//==================================================================================================
//								RJM Maszyny sp. z o.o.
//									04.02.2022
//	Obsługa elektrozaworu 5/3 odpowietrzony w pozycji środkowej
// 	v1.0	|| TC v 3.1.4024.22		|| - pierwsza wersja
//==================================================================================================
FUNCTION_BLOCK FB_Elektrozawor_5na3_Odpowietrzony IMPLEMENTS I_Elektrozawor_5na
VAR
	fbCewkaA								: FB_ElektrozaworCewka;
	fbCewkaB								: FB_ElektrozaworCewka;
END_VAR

//==================================================================================================
//								RJM Maszyny sp. z o.o.
//									04.02.2022
//	Włączenie cewki - wyjscie 2
// 	v1.0	|| TC v 3.1.4024.22		|| - pierwsza wersja
//==================================================================================================METHOD WlaczWyjscie2 : BOOL
VAR_INPUT
END_VAR
fbCewkaA.Wlacz ();
END_METHOD

//==================================================================================================
//								RJM Maszyny sp. z o.o.
//									04.02.2022
//	Włączenie cewki - wyjscie 4
// 	v1.0	|| TC v 3.1.4024.22		|| - pierwsza wersja
//==================================================================================================
METHOD WlaczWyjscie4 : BOOL
VAR_INPUT
END_VAR
fbCewkaB.Wlacz ();
END_METHOD

//==================================================================================================
//								RJM Maszyny sp. z o.o.
//									04.02.2022
//	Wyłączenie cewki - wyjscie 2
// 	v1.0	|| TC v 3.1.4024.22		|| - pierwsza wersja
//==================================================================================================METHOD WylaczWyjscie2 : BOOL
VAR_INPUT
END_VAR
fbCewkaA.Wylacz ();
END_METHOD

//==================================================================================================
//								RJM Maszyny sp. z o.o.
//									04.02.2022
//	Wyłączenie cewki - wyjscie 4
// 	v1.0	|| TC v 3.1.4024.22		|| - pierwsza wersja
//==================================================================================================
METHOD WylaczWyjscie4 : BOOL
VAR_INPUT
END_VAR
fbCewkaB.Wylacz ();
END_METHOD

END_FUNCTION_BLOCK

(* stored: Version 1.1.0.1, ProductVersion 3.1.4024.11
   POU FB_Elektrozawor_5na3_Odpowietrzony: Id {f17b99e1-6967-4370-8cd2-c2384288e58c}, SpecialFunc None
   Method WlaczWyjscie2: Id {05977016-e664-463d-87c0-181849a20e65}
   Method WlaczWyjscie4: Id {cc4e5290-0150-4cef-b5cd-45f8eb479fdd}
   Method WylaczWyjscie2: Id {6db52a01-b744-4f16-808b-326aaf1d575a}
   Method WylaczWyjscie4: Id {e3696199-e3d2-4c52-a5b4-578b6fa733f5} *)
